(* Logix 5000 project; controller CeramicPress Emulate 5570 rev 30.12; software revision 30.00 *)

TASK MainTask (continuous, watchdog 500 ms) : MainProgram

MODULES
   Local : Emulate 5570 (ICP 2, rev 30.12)
END_MODULES

VAR_GLOBAL   (* controller tags *)
   ActLX : INT;
   ActLY : INT;
   CilinderMax : BOOL;
   CilinderMin : BOOL;
   CilinderPos : INT;
   FillerMax : BOOL;
   FillerMin : BOOL;
   FillerPos : INT;
   Manguera : BOOL;
   PosLX : INT;
   PosLY : INT;
   SourceTiles : BOOL;
   Start : BOOL;
   StartPress : BOOL;
   SXmax : BOOL;
   SXmin : BOOL;
   TileMax : BOOL;
   TileMin : BOOL;
   TilePos : INT;
   Tipper_Grab : INT;
   Tipper_Rollers : BOOL := 1;
   Tipper_Rotate : INT;
   Tipper_S1 : BOOL;
   Tipper_S2 : BOOL;
   VelX : INT;
   VelY : INT;
   Xmax : BOOL;
   Xmin : BOOL;
   Ymax : BOOL;
   Ymin : BOOL;
END_VAR

PROGRAM MainProgram   (* main routine MainRoutine *)
VAR
   Action_000 : SFC_ACTION := (Status := 16#c020_0000, A := 1, Q := 1, PauseTimer := 1, Count := 7);
   Action_001 : SFC_ACTION := (Status := 16#0020_0000, PauseTimer := 1);
   Action_002 : SFC_ACTION := (Status := 16#0020_0000, PauseTimer := 1);
   Action_003 : SFC_ACTION := (Status := 16#0020_0000, PauseTimer := 1);
   Action_004 : SFC_ACTION := (Status := 16#0020_0000, PauseTimer := 1);
   Action_005 : SFC_ACTION := (Status := 16#0020_0000, PauseTimer := 1);
   Action_006 : SFC_ACTION := (Status := 16#0020_0000, PauseTimer := 1);
   Action_007 : SFC_ACTION := (Status := 16#0020_0000, PauseTimer := 1);
   Action_008 : SFC_ACTION := (Status := 16#0020_0000, PauseTimer := 1);
   Action_009 : SFC_ACTION := (Status := 16#0020_0000, PauseTimer := 1);
   Action_010 : SFC_ACTION := (Status := 16#0020_0000, PauseTimer := 1);
   Action_011 : SFC_ACTION := (Status := 16#0020_0000, PauseTimer := 1);
   Action_012 : SFC_ACTION := (Status := 16#0020_0000, PauseTimer := 1);
   Action_013 : SFC_ACTION := (Status := 16#0020_0000, PauseTimer := 1);
   Action_014 : SFC_ACTION := (Status := 16#0020_0000, PauseTimer := 1, PRE := 2000);
   Action_015 : SFC_ACTION := (Status := 16#0020_0000, PauseTimer := 1);
   Action_016 : SFC_ACTION := (Status := 16#0020_0000, PauseTimer := 1);
   Action_017 : SFC_ACTION := (Status := 16#0020_0000, PauseTimer := 1, Count := 5);
   Action_018 : SFC_ACTION := (Status := 16#0020_0000, PauseTimer := 1, Count := 5);
   Action_019 : SFC_ACTION := (Status := 16#0020_0000, PauseTimer := 1, Count := 5);
   Action_020 : SFC_ACTION := (Status := 16#0020_0000, PauseTimer := 1, Count := 5);
   Action_021 : SFC_ACTION := (Status := 16#0020_0000, PauseTimer := 1, Count := 5);
   Action_022 : SFC_ACTION := (Status := 16#0020_0000, PauseTimer := 1, Count := 1);
   Action_023 : SFC_ACTION := (Status := 16#0020_0000, PauseTimer := 1, Count := 1);
   Action_024 : SFC_ACTION := (Status := 16#0020_0000, PauseTimer := 1, Count := 1);
   Action_025 : SFC_ACTION := (Status := 16#0020_0000, PauseTimer := 1, Count := 1);
   Action_026 : SFC_ACTION := (Status := 16#0020_0000, PauseTimer := 1, Count := 1);
   Action_027 : SFC_ACTION := (Status := 16#0020_0000, PauseTimer := 1);
   CountSource : COUNTER := (PRE := 1);
   Step_000 : SFC_STEP := (Status := 16#0020_0000, PauseTimer := 1);
   Step_001 : SFC_STEP := (Status := 16#0020_0001, PauseTimer := 1);   // Mover hopper en x+
   Step_002 : SFC_STEP := (Status := 16#0020_0000, PauseTimer := 1);
   Step_003 : SFC_STEP := (Status := 16#0020_0000, PauseTimer := 1);   // Mover hopper en x-
   Step_004 : SFC_STEP := (Status := 16#0020_0000, PauseTimer := 1);
   Step_005 : SFC_STEP := (Status := 16#0020_0000, PauseTimer := 1);
   Step_006 : SFC_STEP := (Status := 16#0020_0000, PauseTimer := 1);
   Step_007 : SFC_STEP := (Status := 16#0020_0000, PauseTimer := 1);
   Step_008 : SFC_STEP := (Status := 16#0020_0000, PauseTimer := 1, PRE := 200);
   Step_009 : SFC_STEP := (Status := 16#0020_0000, PauseTimer := 1);
   Step_010 : SFC_STEP := (Status := 16#0020_0001, PauseTimer := 1);
   Step_011 : SFC_STEP := (Status := 16#0020_0001, PauseTimer := 1);
   Step_012 : SFC_STEP := (Status := 16#0020_0000, PauseTimer := 1);
   Step_013 : SFC_STEP := (Status := 16#0020_0201, PauseTimer := 1);
   Step_014 : SFC_STEP := (Status := 16#0020_0001, PauseTimer := 1);
   Step_015 : SFC_STEP := (Status := 16#0820_0201, DN := 1, PauseTimer := 1, T := 20, TMax := 20, Count := 1);
   Step_016 : SFC_STEP := (Status := 16#0020_0001, PauseTimer := 1);
   Step_017 : SFC_STEP := (Status := 16#0020_0001, PauseTimer := 1);
   Step_018 : SFC_STEP := (Status := 16#0020_0001, PauseTimer := 1);
   Step_019 : SFC_STEP := (Status := 16#0020_0001, PauseTimer := 1);
   Step_020 : SFC_STEP := (Status := 16#0020_0001, PauseTimer := 1);
   Step_021 : SFC_STEP := (Status := 16#0020_0001, PauseTimer := 1);
   Step_022 : SFC_STEP := (Status := 16#0020_0001, PauseTimer := 1);
   Step_023 : SFC_STEP := (Status := 16#0020_0001, PauseTimer := 1);
   Step_024 : SFC_STEP := (Status := 16#0020_0001, PauseTimer := 1);
   Step_025 : SFC_STEP := (Status := 16#0020_0001, PauseTimer := 1);
   Step_026 : SFC_STEP := (Status := 16#0020_0001, PauseTimer := 1);
   Step_027 : SFC_STEP := (Status := 16#0020_0000, PauseTimer := 1);
   Step_028 : SFC_STEP := (Status := 16#a820_0001, X := 1, SA := 1, DN := 1, PauseTimer := 1, T := 149836, TMax := 149836, Count := 7);
   Step_029 : SFC_STEP := (Status := 16#0820_0001, DN := 1, PauseTimer := 1, PRE := 500, T := 579, TMax := 589, Count := 5);
   Step_030 : SFC_STEP := (Status := 16#0020_0001, PauseTimer := 1);
   Step_031 : SFC_STEP := (Status := 16#0020_0001, PauseTimer := 1);
   Step_032 : SFC_STEP := (Status := 16#0820_0001, DN := 1, PauseTimer := 1, PRE := 500, T := 550, TMax := 562, Count := 5);
   Step_033 : SFC_STEP := (Status := 16#0820_0001, DN := 1, PauseTimer := 1, PRE := 500, T := 575, TMax := 583, Count := 5);
   Step_034 : SFC_STEP := (Status := 16#0820_0001, DN := 1, PauseTimer := 1, PRE := 1000, T := 1027, TMax := 1046, Count := 5);
   Step_035 : SFC_STEP := (Status := 16#0820_0001, DN := 1, PauseTimer := 1, T := 22, TMax := 26, Count := 5);
   Step_036 : SFC_STEP := (Status := 16#0020_0001, PauseTimer := 1, PRE := 500, T := 24, TMax := 24, Count := 1);
   Step_037 : SFC_STEP := (Status := 16#0020_0001, PauseTimer := 1, PRE := 500, T := 23, TMax := 23, Count := 1);
   Step_038 : SFC_STEP := (Status := 16#0020_0001, PauseTimer := 1, PRE := 500, T := 26, TMax := 26, Count := 1);
   Step_039 : SFC_STEP := (Status := 16#0020_0001, PauseTimer := 1, PRE := 1000, T := 22, TMax := 22, Count := 1);
   Step_040 : SFC_STEP := (Status := 16#0020_0001, PauseTimer := 1);
   Step_041 : SFC_STEP := (Status := 16#0020_0001, PauseTimer := 1);
   Step_042 : SFC_STEP := (Status := 16#0020_0001, PauseTimer := 1);
   Step_043 : SFC_STEP := (Status := 16#0820_0001, DN := 1, PauseTimer := 1, T := 22, TMax := 22, Count := 1);
   Step_044 : SFC_STEP := (Status := 16#0820_0001, DN := 1, PauseTimer := 1, T := 68, TMax := 68, Count := 6);
   Step_045 : SFC_STEP := (Status := 16#0020_0000, PauseTimer := 1);
   Step_046 : SFC_STEP := (Status := 16#0020_0000, PauseTimer := 1);
   Step_050 : SFC_STEP := (Status := 16#0020_0000, PauseTimer := 1, PRE := 200);
   Step_051 : SFC_STEP := (Status := 16#0020_0001, PauseTimer := 1, PRE := 200);
   Timer1 : TIMER := (PRE := 41);
   Tran_000 : BOOL;
   Tran_001 : BOOL;
   Tran_002 : BOOL;
   Tran_003 : BOOL;
   Tran_004 : BOOL;
   Tran_005 : BOOL;
   Tran_006 : BOOL;
   Tran_007 : BOOL;
   Tran_008 : BOOL;
   Tran_009 : BOOL := 1;
   Tran_010 : BOOL;
   Tran_011 : BOOL;
   Tran_012 : BOOL;
   Tran_013 : BOOL;
   Tran_014 : BOOL;
   Tran_015 : BOOL;
   Tran_016 : BOOL;
   Tran_017 : BOOL;
   Tran_018 : BOOL;
   Tran_019 : BOOL;
   Tran_020 : BOOL;
   Tran_021 : BOOL := 1;
   Tran_022 : BOOL;
   Tran_023 : BOOL := 1;
   Tran_024 : BOOL := 1;
   Tran_025 : BOOL := 1;
   Tran_026 : BOOL := 1;
   Tran_027 : BOOL := 1;
   Tran_028 : BOOL := 1;
   Tran_029 : BOOL;
   Tran_030 : BOOL := 1;
   Tran_031 : BOOL := 1;
   Tran_032 : BOOL := 1;
   Tran_033 : BOOL := 1;
   Tran_034 : BOOL := 1;
   Tran_035 : BOOL;
   Tran_036 : BOOL;
END_VAR

ROUTINE MainRoutine   (* ladder *)
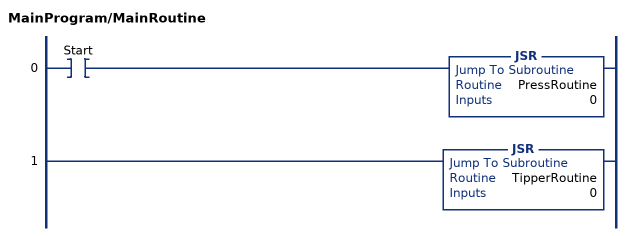
   0: XIC(Start)JSR(PressRoutine,0);
   1: JSR(TipperRoutine,0);
END_ROUTINE

ROUTINE PressRoutine   (* sequential function chart *)
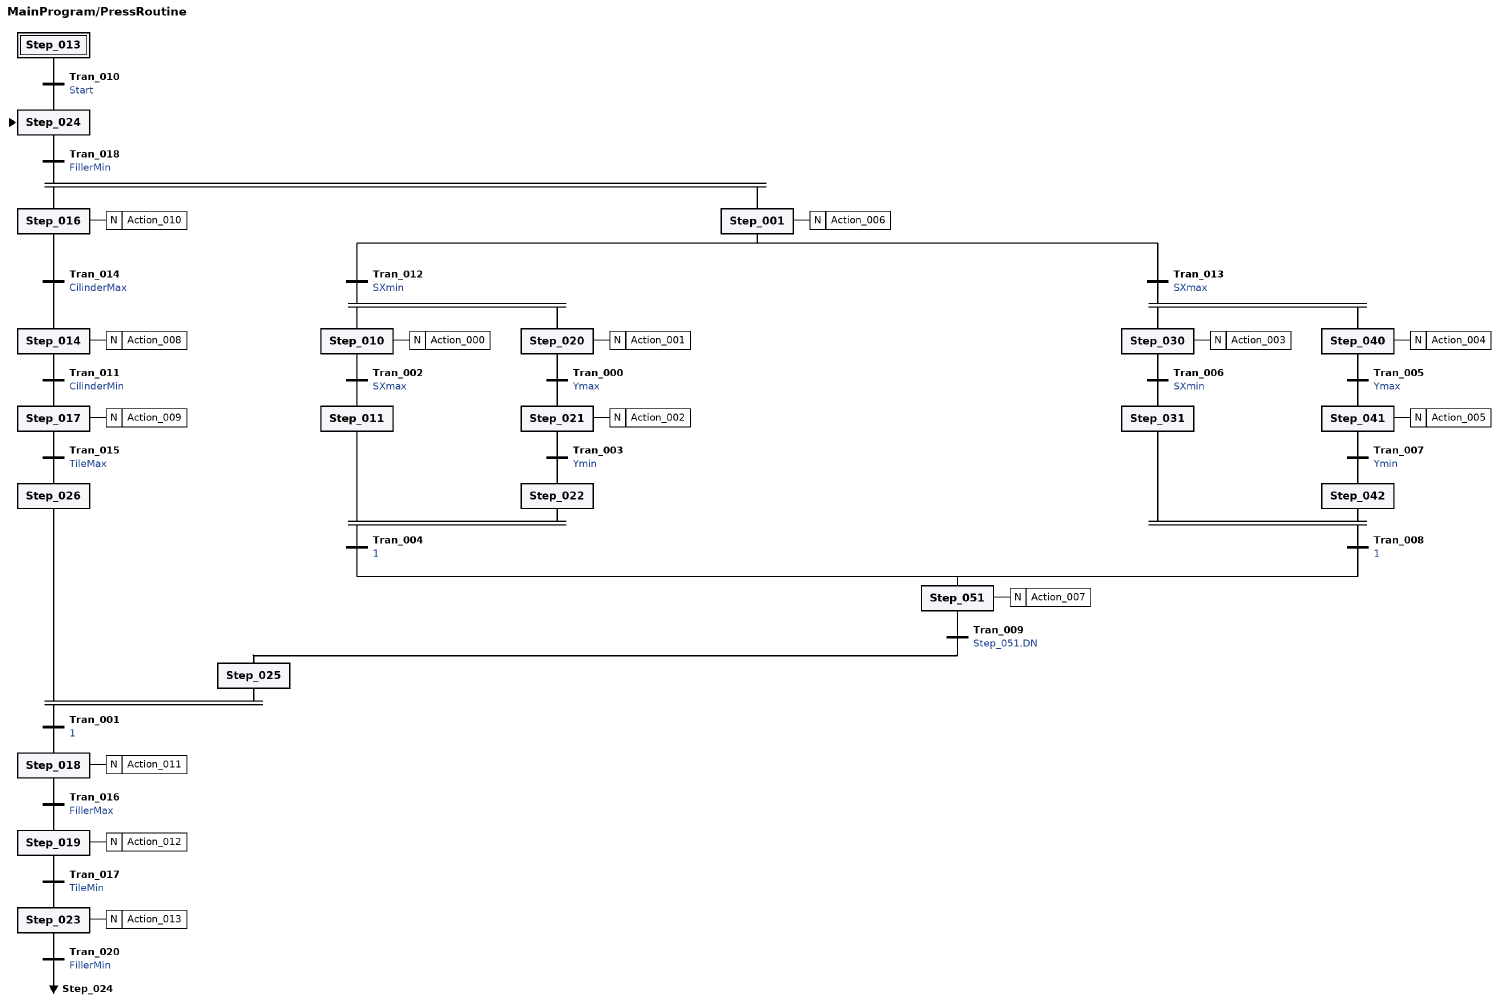
   INITIAL_STEP Step_013:
   END_STEP
   TRANSITION Tran_010 FROM Step_013 TO Step_024
      := Start
   END_TRANSITION
   STEP Step_024:
   END_STEP
   TRANSITION Tran_018 FROM Step_024 TO (Step_016, Step_001)
      := FillerMin
   END_TRANSITION
   STEP Step_016:
      ACTION Action_010 (N):
         CilinderPos := 140;
         SourceTiles :=1;
      END_ACTION
   END_STEP
   STEP Step_001:
      ACTION Action_006 (N):
         Manguera :=1;
      END_ACTION
   END_STEP
   TRANSITION Tran_014 FROM Step_016 TO Step_014
      := CilinderMax
   END_TRANSITION
   TRANSITION Tran_012 FROM Step_001 TO (Step_020, Step_010)
      := SXmin
   END_TRANSITION
   TRANSITION Tran_013 FROM Step_001 TO (Step_040, Step_030)
      := SXmax
   END_TRANSITION
   STEP Step_014:
      ACTION Action_008 (N):
         SourceTiles :=0;
         CilinderPos := 0;
         
      END_ACTION
   END_STEP
   TRANSITION Tran_011 FROM Step_014 TO Step_017
      := CilinderMin
         
   END_TRANSITION
   STEP Step_010:
      ACTION Action_000 (N):
         ActLX := 1220;
      END_ACTION
   END_STEP
   STEP Step_020:
      ACTION Action_001 (N):
         ActLY := 710;
      END_ACTION
   END_STEP
   STEP Step_017:
      ACTION Action_009 (N):
         TilePos := 9;
      END_ACTION
   END_STEP
   STEP Step_030:
      ACTION Action_003 (N):
         ActLX := 0;
      END_ACTION
   END_STEP
   STEP Step_040:
      ACTION Action_004 (N):
         ActLY := 710;
      END_ACTION
   END_STEP
   TRANSITION Tran_002 FROM Step_010 TO Step_011
      := SXmax
   END_TRANSITION
   TRANSITION Tran_000 FROM Step_020 TO Step_021
      := Ymax
   END_TRANSITION
   TRANSITION Tran_015 FROM Step_017 TO Step_026
      := TileMax
         
   END_TRANSITION
   TRANSITION Tran_006 FROM Step_030 TO Step_031
      := SXmin
   END_TRANSITION
   TRANSITION Tran_005 FROM Step_040 TO Step_041
      := Ymax
   END_TRANSITION
   STEP Step_021:
      ACTION Action_002 (N):
         ActLY := 0;
         
      END_ACTION
   END_STEP
   STEP Step_026:
   END_STEP
   STEP Step_025:
   END_STEP
   STEP Step_041:
      ACTION Action_005 (N):
         ActLY := 0;
      END_ACTION
   END_STEP
   TRANSITION Tran_003 FROM Step_021 TO Step_022
      := Ymin
   END_TRANSITION
   TRANSITION Tran_007 FROM Step_041 TO Step_042
      := Ymin
   END_TRANSITION
   TRANSITION Tran_001 FROM (Step_025, Step_026) TO Step_018
      := 1
   END_TRANSITION
   STEP Step_011:
   END_STEP
   STEP Step_022:
   END_STEP
   STEP Step_031:
   END_STEP
   STEP Step_042:
   END_STEP
   STEP Step_018:
      ACTION Action_011 (N):
         FillerPos := 800;
      END_ACTION
   END_STEP
   TRANSITION Tran_004 FROM (Step_011, Step_022) TO Step_051
      := 1
   END_TRANSITION
   TRANSITION Tran_008 FROM (Step_031, Step_042) TO Step_051
      := 1
   END_TRANSITION
   TRANSITION Tran_016 FROM Step_018 TO Step_019
      := FillerMax
   END_TRANSITION
   STEP Step_019:
      ACTION Action_012 (N):
         TilePos := 0;
      END_ACTION
   END_STEP
   STEP Step_051:
      ACTION Action_007 (N):
         Manguera :=0;
      END_ACTION
   END_STEP
   TRANSITION Tran_017 FROM Step_019 TO Step_023
      := TileMin
         
   END_TRANSITION
   TRANSITION Tran_009 FROM Step_051 TO Step_025
      := Step_051.DN
   END_TRANSITION
   STEP Step_023:
      ACTION Action_013 (N):
         FillerPos := 0;
      END_ACTION
   END_STEP
   TRANSITION Tran_020 FROM Step_023 TO Step_024
      := FillerMin
         
   END_TRANSITION
END_ROUTINE

ROUTINE TipperRoutine   (* sequential function chart *)
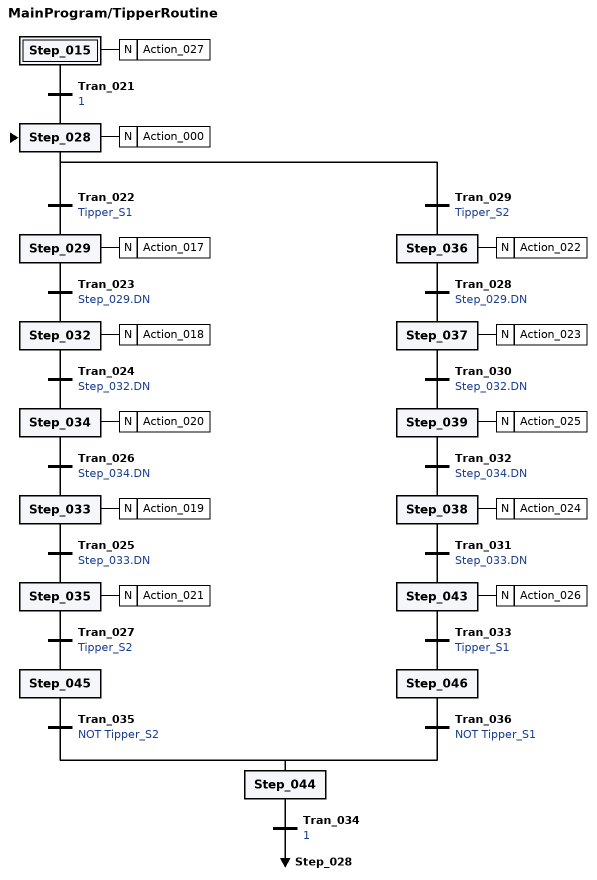
   INITIAL_STEP Step_015:
      ACTION Action_027 (N):
         Tipper_Rotate :=0;
      END_ACTION
   END_STEP
   TRANSITION Tran_021 FROM Step_015 TO Step_028
      := 1
         
   END_TRANSITION
   STEP Step_028:
      ACTION Action_000 (N):
         Tipper_Rollers :=1;
      END_ACTION
   END_STEP
   TRANSITION Tran_022 FROM Step_028 TO Step_029
      := Tipper_S1
   END_TRANSITION
   TRANSITION Tran_029 FROM Step_028 TO Step_036
      := Tipper_S2
         
   END_TRANSITION
   STEP Step_029:
      ACTION Action_017 (N):
         Tipper_Rollers :=0;
      END_ACTION
   END_STEP
   STEP Step_036:
      ACTION Action_022 (N):
         Tipper_Rollers :=0;
      END_ACTION
   END_STEP
   TRANSITION Tran_023 FROM Step_029 TO Step_032
      := Step_029.DN
   END_TRANSITION
   TRANSITION Tran_028 FROM Step_036 TO Step_037
      := Step_029.DN
   END_TRANSITION
   STEP Step_032:
      ACTION Action_018 (N):
         Tipper_Grab:=10;
      END_ACTION
   END_STEP
   STEP Step_037:
      ACTION Action_023 (N):
         Tipper_Grab:=10;
      END_ACTION
   END_STEP
   TRANSITION Tran_024 FROM Step_032 TO Step_034
      := Step_032.DN
   END_TRANSITION
   TRANSITION Tran_030 FROM Step_037 TO Step_039
      := Step_032.DN
   END_TRANSITION
   STEP Step_034:
      ACTION Action_020 (N):
         Tipper_Rotate:=180;
      END_ACTION
   END_STEP
   STEP Step_039:
      ACTION Action_025 (N):
         Tipper_Rotate:=0;
      END_ACTION
   END_STEP
   TRANSITION Tran_026 FROM Step_034 TO Step_033
      := Step_034.DN
   END_TRANSITION
   TRANSITION Tran_032 FROM Step_039 TO Step_038
      := Step_034.DN
   END_TRANSITION
   STEP Step_033:
      ACTION Action_019 (N):
         Tipper_Grab :=0;
      END_ACTION
   END_STEP
   STEP Step_038:
      ACTION Action_024 (N):
         Tipper_Grab :=0;
      END_ACTION
   END_STEP
   TRANSITION Tran_025 FROM Step_033 TO Step_035
      := Step_033.DN
   END_TRANSITION
   TRANSITION Tran_031 FROM Step_038 TO Step_043
      := Step_033.DN
   END_TRANSITION
   STEP Step_035:
      ACTION Action_021 (N):
         Tipper_Rollers :=1;
      END_ACTION
   END_STEP
   STEP Step_043:
      ACTION Action_026 (N):
         Tipper_Rollers :=1;
      END_ACTION
   END_STEP
   TRANSITION Tran_027 FROM Step_035 TO Step_045
      := Tipper_S2
   END_TRANSITION
   TRANSITION Tran_033 FROM Step_043 TO Step_046
      := Tipper_S1
   END_TRANSITION
   STEP Step_045:
   END_STEP
   STEP Step_046:
   END_STEP
   TRANSITION Tran_035 FROM Step_045 TO Step_044
      := NOT Tipper_S2
   END_TRANSITION
   TRANSITION Tran_036 FROM Step_046 TO Step_044
      := NOT Tipper_S1
   END_TRANSITION
   STEP Step_044:
   END_STEP
   TRANSITION Tran_034 FROM Step_044 TO Step_028
      := 1
   END_TRANSITION
END_ROUTINE
END_PROGRAM
